Staubli VAL3: saveIt.pgx

program saveIt(bool& x_bSave[] (dimensions=1))
  local string l_sMessage
  local num l_nResult
  local string l_sResult
begin
  // unselect ALL
  call unSelectItem()
  // do the onSave trajtype
  l_sResult=""
  call trajType:onSave(l_sResult)
  //
  if l_nResult==0
    logMsg("[KERNEL] INTERFACE:Save the trajectory "+saveData:sTrajTypeUsing+": "+sTrajName)
    x_bSave=false
    call language:message(l_sMessage,-4)
    call use:timerDialog(l_sMessage,1)
  else
    popUpMsg("Save code error "+toString("",l_nResult))
  endIf
end
